FUNCTION_BLOCK strip_set_pixel (* Service Interface Function Block Type *)
  (* Standard: 61499-2; Description: Copyright (c) 2022 HR Agrartechnik GmbH This program and the accompanying materials are made available under the terms of the Eclipse Public License 2.0 which is available at https://www.eclipse.org/legal/epl-2.0/ SPDX-License-Identifier: EPL-2.0 *)
  (* Version 1.0, 2022-07-16, franz *)
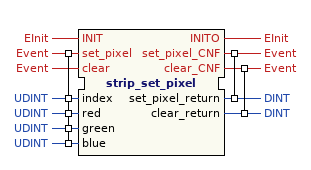
  EVENT_INPUT
    INIT : EInit; (* Service Initialization *)
    set_pixel WITH index, red, green, blue; (* Set RGB for a specific pixel *)
    clear; (* Clear LED strip (turn off all LEDs) *)
  END_EVENT
  EVENT_OUTPUT
    INITO : EInit; (* Initialization Confirm *)
    set_pixel_CNF WITH set_pixel_return; (* Confirmation of set_pixel *)
    clear_CNF WITH clear_return; (* Confirmation of clear *)
  END_EVENT
  VAR_INPUT
    index : UDINT; (* index of pixel to set *)
    red : UDINT; (* red part of color *)
    green : UDINT; (* green part of color *)
    blue : UDINT; (* blue part of color *)
  END_VAR
  VAR_OUTPUT
    set_pixel_return : DINT; (* Error indication *)
    clear_return : DINT;
  END_VAR
END_FUNCTION_BLOCK
